ABB RAPID module: HandEyeCalibrationExample.modx

MODULE RcHandEyeCalibrationExample
    ! Hand-Eye Calibration Example Module
    ! This module demonstrates how to perform hand-eye calibration with the Roboception system.
    ! The calibration requires at least 8 distinct robot poses where the calibration grid
    ! is fully visible to the camera from different angles and positions.
    ! For detailed guidance on optimal calibration poses, refer to:
    ! https://doc.rc-cube.com/latest/en/handeye_calibration.html#step-3-record-poses

    ! Pipeline ID for hand-eye calibration
    CONST num HEC_PIPELINE_ID := 1;

    ! Calibration poses - these should be different robot poses that:
    ! 1. Give good coverage of the workspace
    ! 2. Provide different viewing angles of the calibration grid
    ! 3. Ensure the calibration grid is fully visible in each pose
    CONST robtarget CAL_POSE_1 := [[232.4,382.9,885.4],[-0.815,0.568,-0.012,0.116],[0,0,0,0],[9E+09,9E+09,9E+09,9E+09,9E+09,9E+09]];
    CONST robtarget CAL_POSE_2 := [[516.7,373.8,676.2],[0.794,-0.579,-0.181,0.022],[0,0,0,0],[9E+09,9E+09,9E+09,9E+09,9E+09,9E+09]];
    CONST robtarget CAL_POSE_3 := [[-214.2,373.8,676.4],[-0.771,0.505,-0.263,0.285],[0,0,0,0],[9E+09,9E+09,9E+09,9E+09,9E+09,9E+09]];
    CONST robtarget CAL_POSE_4 := [[218.6,629.9,676.1],[0.816,-0.574,0.047,0.048],[0,0,0,0],[9E+09,9E+09,9E+09,9E+09,9E+09,9E+09]];
    CONST robtarget CAL_POSE_5 := [[312.8,409.0,408.6],[-0.816,0.575,0.019,0.046],[0,0,0,0],[9E+09,9E+09,9E+09,9E+09,9E+09,9E+09]];
    CONST robtarget CAL_POSE_6 := [[645.4,409.2,335.7],[0.777,-0.565,-0.252,0.121],[0,0,0,0],[9E+09,9E+09,9E+09,9E+09,9E+09,9E+09]];
    CONST robtarget CAL_POSE_7 := [[-39.2,409.3,328.5],[-0.763,0.515,-0.292,0.261],[0,0,0,0],[9E+09,9E+09,9E+09,9E+09,9E+09,9E+09]];
    CONST robtarget CAL_POSE_8 := [[291.2,610.4,328.0],[0.796,-0.548,0.173,0.193],[0,0,0,0],[9E+09,9E+09,9E+09,9E+09,9E+09,9E+09]];

    PROC perform_hand_eye_calibration()
        ! Initialize HEC pipeline
        IF NOT hec_init(HEC_PIPELINE_ID \debug:=TRUE) THEN
            ErrWrite \W, "HECError", "Failed to initialize hand-eye calibration";
            RETURN;
        ENDIF

        ! Move to and collect data for each calibration pose
        IF NOT collect_calibration_pose(1, CAL_POSE_1) THEN
            RETURN;
        ENDIF

        IF NOT collect_calibration_pose(2, CAL_POSE_2) THEN
            RETURN;
        ENDIF

        IF NOT collect_calibration_pose(3, CAL_POSE_3) THEN
            RETURN;
        ENDIF

        IF NOT collect_calibration_pose(4, CAL_POSE_4) THEN
            RETURN;
        ENDIF

        IF NOT collect_calibration_pose(5, CAL_POSE_5) THEN
            RETURN;
        ENDIF

        IF NOT collect_calibration_pose(6, CAL_POSE_6) THEN
            RETURN;
        ENDIF

        IF NOT collect_calibration_pose(7, CAL_POSE_7) THEN
            RETURN;
        ENDIF

        IF NOT collect_calibration_pose(8, CAL_POSE_8) THEN
            RETURN;
        ENDIF

        ! Perform final calibration calculation
        IF NOT hec_calibrate(HEC_PIPELINE_ID \debug:=TRUE) THEN
            ErrWrite \W, "HECError", "Failed to perform calibration";
            RETURN;
        ENDIF

        ErrWrite \I, "HECSuccess", "Hand-eye calibration completed successfully";

    ERROR
        ErrWrite \W, "HECError", "Error during hand-eye calibration: " + NumToStr(ERRNO, 0);
    ENDPROC

    ! Helper function to move to a pose and collect calibration data
    FUNC bool collect_calibration_pose(num pose_num, robtarget target)
        ! Move to calibration pose with high precision
        MoveJ target, v50, fine, tool0;

        ! Wait for robot to settle
        WaitTime 1;

        ! Set the pose for calibration
        IF NOT hec_set_pose(HEC_PIPELINE_ID, pose_num, target \debug:=TRUE) THEN
            ErrWrite \W, "HECError", "Failed to set pose " + NumToStr(pose_num, 0);
            RETURN FALSE;
        ENDIF

        RETURN TRUE;

    ERROR
        ErrWrite \W, "HECError", "Error collecting pose " + NumToStr(pose_num, 0) + ": " + NumToStr(ERRNO, 0);
        RETURN FALSE;
    ENDFUNC

ENDMODULE
